Fanuc KAREL source: NC0063.KL

-- PROVISIONAL review KL for V1013-1; original PC SHA256 3c65e78651fa3cc679c181e22c71d99d2ca74921126bd542cd26e1fc689ecc9a
-- Incomplete behavior may be omitted. Consult companion uncertainty JSON. Do not deploy.
PROGRAM NC0063
%NOLOCKGROUP
-- UNRESOLVED_LOCAL_POOL 3 cells at code offset 3; source declarations unknown
-- DIRECT_LOCAL_WORD_ACCESS alone does not prove INTEGER, REAL, or BOOLEAN
BEGIN
  -- UNRESOLVED_PC offsets 0-8; opcodes 2B,2C,7B
  -- UNRESOLVED_PC offsets 13-20; opcodes 9D,23
  -- UNRESOLVED_PC offsets 25-54; opcodes 9D,23,9E,2E,22,7A
  -- UNRESOLVED_PC offsets 59-88; opcodes 9D,23,9E,2E,22,7A
  -- UNRESOLVED_PC offsets 93-107; opcodes 21,9D,52,23
  -- UNRESOLVED_PC offsets 112-127; opcodes 20,2C,23
  -- UNRESOLVED_PC offsets 132-147; opcodes 20,2C,23
  -- UNRESOLVED_PC offsets 152-156; opcodes 7F
  -- UNRESOLVED_PC offsets 161-165; opcodes 27,AA
  -- UNRESOLVED_PC offsets 170-174; opcodes 7F
END NC0063
